Fanuc KAREL source: app_check.kl

PROGRAM appcheck
%COMMENT = 'appcheck v1'
%NOLOCKGROUP
%NOPAUSE=ERROR+COMMAND+TPENABLE
%NOBUSYLAMP

CONST

	PR_JOINTS = 40
	PR_XYZWPR = 41

	R_KEEP = 42

	R_XMAX = 43
	R_YMAX = 44
	R_ZMAX = 45
	R_XMIN = 46
	R_YMIN = 47
	R_ZMIN = 48

	R_COORD1 = 51
	R_COORD2 = 52
	R_COORD3 = 53
	R_COORD4 = 54
	R_COORD5 = 55
	R_COORD6 = 56

VAR

	STATUS: INTEGER

	cur_pos: XYZWPR
	new_jpos: JOINTPOS
	new_pos: XYZWPREXT

	reach_ab: INTEGER

	limit_x: INTEGER
	limit_y: INTEGER
	limit_z: INTEGER

	config_ref: INTEGER
	out_pos: POSITION
	wjnt_cfg: CONFIG
	ext_ang: ARRAY[3] OF REAL

	keep_flag: BOOLEAN

	keep_int: INTEGER

	keep_real: REAL

	xmax_flag: BOOLEAN
	ymax_flag: BOOLEAN
	zmax_flag: BOOLEAN
	xmin_flag: BOOLEAN
	ymin_flag: BOOLEAN
	zmin_flag: BOOLEAN

	xmax_int: INTEGER
	ymax_int: INTEGER
	zmax_int: INTEGER
	xmin_int: INTEGER
	ymin_int: INTEGER
	zmin_int: INTEGER

	xmax_real: REAL
	ymax_real: REAL
	zmax_real: REAL
	xmin_real: REAL
	ymin_real: REAL
	zmin_real: REAL

ROUTINE checkLimit

BEGIN

	--limit the XYZ direction

	IF xmin_flag THEN
		IF new_pos.x <= xmin_real THEN
			FLG[8] = ON
			limit_x = 6
		ENDIF
	ELSE
		IF new_pos.x <= xmin_int THEN
			FLG[8] = ON
			limit_x = 6
		ENDIF
	ENDIF

	IF xmax_flag THEN
		IF new_pos.x >= xmax_real THEN
			FLG[8] = ON
			limit_x = 3
		ENDIF
	ELSE
		IF new_pos.x >= xmax_int THEN
			FLG[8] = ON
			limit_x = 3
		ENDIF
	ENDIF

	IF ymin_flag THEN
		IF new_pos.y <= ymin_real THEN
			FLG[8] = ON
			limit_y = 6
		ENDIF
	ELSE
		IF new_pos.y <= ymin_int THEN
			FLG[8] = ON
			limit_y = 6
		ENDIF
	ENDIF

	IF ymax_flag THEN
		IF new_pos.y >= ymax_real THEN
			FLG[8] = ON
			limit_y = 3
		ENDIF
	ELSE
		IF new_pos.y >= ymax_int THEN
			FLG[8] = ON
			limit_y = 3
		ENDIF
	ENDIF

	IF zmin_flag THEN
		IF new_pos.z <= zmin_real THEN
			FLG[8] = ON
			limit_z = 6
		ENDIF
	ELSE
		IF new_pos.z <= zmin_int THEN
			FLG[8] = ON
			limit_z = 6
		ENDIF
	ENDIF

	IF zmax_flag THEN
		IF new_pos.z >= zmax_real THEN
			FLG[8] = ON
			limit_z = 3
		ENDIF
	ELSE
		IF new_pos.z >= zmax_int THEN
			FLG[8] = ON
			limit_z = 3
		ENDIF
	ENDIF

END checkLimit

BEGIN

	GET_REG(R_KEEP, keep_flag, keep_int, keep_real, STATUS )

	GET_REG(R_XMAX, xmax_flag, xmax_int, xmax_real, STATUS)
	GET_REG(R_YMAX, ymax_flag, ymax_int, ymax_real, STATUS)
	GET_REG(R_ZMAX, zmax_flag, zmax_int, zmax_real, STATUS)
	GET_REG(R_XMIN, xmin_flag, xmin_int, xmin_real, STATUS)
	GET_REG(R_YMIN, ymin_flag, ymin_int, ymin_real, STATUS)
	GET_REG(R_ZMIN, zmin_flag, zmin_int, zmin_real, STATUS)

	reach_ab = 0

	limit_x = 0
	limit_y = 0
	limit_z = 0

	--check the new jpos is in range

	IF FLG[1] OR FLG[2] THEN

		new_jpos = GET_JPOS_REG(PR_JOINTS, STATUS)

		IF (STATUS <> 0 ) THEN

			WRITE ('GET_JPOS_REG  built-IN failed WITH STATUS = ', STATUS, CR)

		ELSE

			IF NOT J_IN_RANGE(new_jpos) THEN
				FLG[8] = ON
				reach_ab = 1
			ELSE
				reach_ab = 0
			ENDIF

			--limit the XYZ direction

			 config_ref = HALF_SOLN

			JOINT2POS (new_jpos, $UFRAME, $UTOOL, config_ref, out_pos, wjnt_cfg, ext_ang, STATUS)

			new_pos = out_pos --Convert out_pos (POSITION) to XYZWPREXT

			checkLimit

		ENDIF

	ENDIF

	--check the new pos is in range

	IF FLG[3] OR FLG[4] OR FLG[5] OR FLG[6] THEN

		new_pos = GET_POS_REG(PR_XYZWPR, STATUS)

		IF (STATUS <> 0 ) THEN

			WRITE ('GET_POS_REG  built-IN failed WITH STATUS = ', STATUS, CR)

		ELSE

			IF NOT IN_RANGE(new_pos) THEN
				FLG[8] = ON
				reach_ab = 1
			ELSE
				reach_ab = 0
			ENDIF

			checkLimit

		ENDIF

	ENDIF

	IF keep_flag THEN
		IF keep_real > 5 THEN
			FLG[8] = ON
		ENDIF
	ELSE
		IF keep_int > 5 THEN
			FLG[8] = ON
		ENDIF
	ENDIF

END appcheck
